(* CODESYS project Estação 5 - Sorting (2022).project

Project tree, tasks and I/O mapping:
  Device : CPX-CEC-C1-V3, Festo AG & Co. KG, order no. 3473128, version 3.5.7.37
      unmapped channels: Rotary switch
    application Application
      libraries: Standard, * (System)
      task MainTask (cyclic, interval t#20ms, priority 20) calls PLC_PRG
      program PLC_PRG [ST]
      global variables GVL
      function ATUALIZAR_VALORES [ST]
      program teste_comunicacao [ST]
      program pisca_pisca [ST]
      function SINALIZAR_QUANTIA_CORES_MODBUS [ST]
    PLC_Diagnosis : PLC-Diagnosis, Festo AG & Co. KG, version 3.5.4.1
    CPX_System : CPX_System, Festo AG & Co. KG, order no. 3473128, version 1.258
      _8DI_8DO_1 : 8DI/8DO, Festo AG & Co. KG, order no. 526257, version 1.258
          settings:  = 0;  = 1;  = 1;  = 1;  = 1;  = 0;  = 1;  = 1;  = 0;  = 0;  = 0;  = 0;  = 0;  = 0;  = 0;  = 0;  = 0;  = 0;  = 0;  = 0;  = 0;  = 0;  = 0;  = 0;  = 0;  = 0;  = 0;  = 0;  = 0;  = 0;  = 0;  = 0;  = 0;  = 0;  = 0;  = 0;  = 0;  = 0;  = 0;  = 0;
             = 0;  = 0;  = 0;  = 0;  = 0;  = 0;  = 0;  = 0;  = 0;  = 0;  = 0;  = 0;  = 0;  = 0;  = 0;  = 0;  = 0;  = 0;  = 0;  = 0;  = 0;  = 0;  = 0;  = 0;  = 0;  = 0;  = 0;  = 0;  = 0;  = 0;  = 0;  = 0;  = 0;  = 0;  = 0;  = 0;  = 0;  = 0;  = 0;  = 0;
             = 576751027668385792;  = 'PI%i.0.0.1=1';  = 'PI%i.0.1.1=1';  = 'PI%i.0.2.1=1';  = 'PI%i.1.0.1=1';  = 'PI%i.1.1.1=0';  = 'PI%i.1.4.2=1';  = 'PI%i.1.6.2=1';  = 'PI%i.6.0.1=0';  = 'PI%i.6.1.1=0';  = 'PI%i.6.2.1=0';  = 'PI%i.6.3.1=0';  = 'PI%i.6.4.1=0';  = 'PI%i.6.5.1=0';  = 'PI%i.6.6.1=0';  = 'PI%i.6.7.1=0';  = dd4a6e61;  = 6
          unmapped channels: Input 0, Output 0
      CEC_C1_V3 : CEC-C1-V3, Festo AG & Co. KG, order no. 3473128, version 1.258
          settings:  = 0;  = 150810762677760;  = 839035072;  = 65535;  = 16885952;  = 13959208;  = 1f5d2989;  = 5
      _8DI_8DO : 8DI/8DO, Festo AG & Co. KG, order no. 526257, version 1.258
          settings:  = 0;  = 1;  = 1;  = 1;  = 1;  = 0;  = 1;  = 1;  = 0;  = 0;  = 0;  = 0;  = 0;  = 0;  = 0;  = 0;  = 0;  = 0;  = 0;  = 0;  = 0;  = 0;  = 0;  = 0;  = 0;  = 0;  = 0;  = 0;  = 0;  = 0;  = 0;  = 0;  = 0;  = 0;  = 0;  = 0;  = 0;  = 0;  = 0;  = 0;
             = 0;  = 0;  = 0;  = 0;  = 0;  = 0;  = 0;  = 0;  = 0;  = 0;  = 0;  = 0;  = 0;  = 0;  = 0;  = 0;  = 0;  = 0;  = 0;  = 0;  = 0;  = 0;  = 0;  = 0;  = 0;  = 0;  = 0;  = 0;  = 0;  = 0;  = 0;  = 0;  = 0;  = 0;  = 0;  = 0;  = 0;  = 0;  = 0;  = 0;
             = 576751027668385792;  = 'PI%i.0.0.1=1';  = 'PI%i.0.1.1=1';  = 'PI%i.0.2.1=1';  = 'PI%i.1.0.1=1';  = 'PI%i.1.1.1=0';  = 'PI%i.1.4.2=1';  = 'PI%i.1.6.2=1';  = 'PI%i.6.0.1=0';  = 'PI%i.6.1.1=0';  = 'PI%i.6.2.1=0';  = 'PI%i.6.3.1=0';  = 'PI%i.6.4.1=0';  = 'PI%i.6.5.1=0';  = 'PI%i.6.6.1=0';  = 'PI%i.6.7.1=0';  = dd4a6e5f;  = 6
          unmapped channels: Input 0, Output 0
    Ethernet : Ethernet, 3S - Smart Software Solutions GmbH, version 3.5.10.0
      ModbusTCP_Slave_Device : ModbusTCP Slave Device, 3S - Smart Software Solutions GmbH, version 3.5.10.0
          unmapped channels: Inputs, Outputs
*)

// Device/Application/GVL
{attribute 'qualified_only'}
VAR_GLOBAL
	//Entradas
	//Sensores
	S_inicio 	AT %IX1.0 :BOOL; //Sensor de inicio da esteira
	S_desv_1 	AT %IX1.1 :BOOL; //Desviacdor 1 avançado
	S_rampa 	AT %IX1.2 :BOOL; //Sensor do fim da esteira
	S_desv_2	AT %IX1.3 :BOOL; //Desviacdor 2 avançado
	S_barreira 	AT %IX1.4  :BOOL; //Sensor de barreira do inicio da esteira
	S_cor 		AT %IX1.5  :BOOL; //Sesnor otico difuso para detectar peças não preta
	S_indutivo  AT %IX1.6  :BOOL; //Sensor indutivo para peças metalicas
	
	//IHM
	Start_btn 		AT	%IX2.0	:BOOL;  //Botão de start
	Stop_btn 		AT	%IX2.1	:BOOL;	//Botão de stop (NF)
	Chave 			AT	%IX2.2	:BOOL;	//Chave auto/manual
	Reset_btn 		AT	%IX2.3	:BOOL;	//Botão de reset
	I4_IHM			AT	%IX2.4	:BOOL;	//Bit de saída 4 da IHM
	I5_IHM			AT	%IX2.5	:BOOL;	//Bit de saída 5 da IHM
	I6_IHM 			AT	%IX2.6	:BOOL;	//Bit de saída 6 da IHM
	I7_IHM			AT	%IX2.7	:BOOL;	//Bit de saída 7 da IHM

//Saídas
	//Atuadorres 			
	Esteira_frente 	AT	%QX0.0	:BOOL;	//Mover a esteira para frente
	Desv_1 			AT	%QX0.1	:BOOL;	//Atua o desviador 1
	Desv_2 	 		AT	%QX0.2	:BOOL;	//Atua o desviador 2
	Stopper		 	AT	%QX0.3	:BOOL;	//Stopper recuado
	//				AT	%QX0.4	:BOOL;	
	//		 		AT	%QX0.5	:BOOL;	
	//				AT	%QX0.6	:BOOL;	
	//	     		AT	%QX0.7	:BOOL;	
	
	//IHM				
	Start_LED		AT	%QX1.0	:BOOL;	//LED do botão de start
	Reset_LED 		AT	%QX1.1	:BOOL;	//LED do botão de reset
	Q1_LED 			AT	%QX1.2	:BOOL;	//LED sinalizador Q1
	Q2_LED			AT	%QX1.3	:BOOL;	//LED sinalizador Q2
	Q4_IHM			AT	%QX1.4	:BOOL;	//Saída Q4 IHM
	Q5_IHM			AT	%QX1.5	:BOOL;	//Saída Q5 IHM
	Q6_IHM			AT	%QX1.6	:BOOL;	//Saída Q6 IHM
	Q7_IHM 			AT	%QX1.7	:BOOL;	//Saída Q7 IHM
	
//MODBUS bits
	//Entradas
	Mod_I_0_0 		AT %IX4.0 : BOOL; //Start 
	Mod_I_0_1	 	AT %IX4.1 : BOOL; //Stop
	Mod_I_0_2 		AT %IX4.2 : BOOL; //Reset
	Mod_I_0_3 		AT %IX4.3 : BOOL; //Modo entrada (DESATIVADO PARA ESSA ESTAÇÃO)
	Mod_I_0_4 		AT %IX4.4 : BOOL; //Modo saída (DESATIVADO PARA ESSA ESTAÇÃO)
	Mod_I_0_5 		AT %IX4.5 : BOOL; //Teste resposta da estação - IN 
	Mod_I_0_6 		AT %IX4.6 : BOOL; //B1 //Confirmação de leitura da informação de peça finalizada pela central
	Mod_I_0_7 		AT %IX4.7 : BOOL; //B2
	Mod_I_1_0 		AT %IX5.0 : BOOL; //B3
	Mod_I_1_1 		AT %IX5.1 : BOOL;
	Mod_I_1_2 		AT %IX5.2 : BOOL;//Confirmação de leitura da informação de peça finalizada pela central
	

	
	//Saídas
	Mod_Q_0_0 		AT %QX2.0 : BOOL; //Estação iniciada							
	Mod_Q_0_1	 	AT %QX2.1 : BOOL; // Estação parada 						
	Mod_Q_0_2 		AT %QX2.2 : BOOL; //Estação em processo										
	Mod_Q_0_3 		AT %QX2.3 : BOOL; // Modo entrada (DESATIVADO PARA ESSA ESTAÇÃO)								
	Mod_Q_0_4 		AT %QX2.4 : BOOL; // Modo saída (DESATIVADO PARA ESSA ESTAÇÃO)
	Mod_Q_0_5 		AT %QX2.5 : BOOL; // Teste resposta da estação - OUT
	
	Mod_Q_0_6 		AT %QX2.6 : BOOL; //B1 														//Sinaliza para a central que uma peça foi finalizada
	
	Mod_Q_0_7 		AT %QX2.7 : BOOL; //B2 														//BLACK B1  LSB
	Mod_Q_1_0 		AT %QX3.0 : BOOL; //B3 														//BLACK B2
	Mod_Q_1_1 		AT %QX3.1 : BOOL; 	   														//BLACK B3  MSB
	
	Mod_Q_1_2 		AT %QX3.2 : BOOL; //Sinaliza para a central que uma peça foi finalizada		//SILVER B1	LSB	
	Mod_Q_1_3 		AT %QX3.3 : BOOL;															//SILVER B2
	Mod_Q_1_4 		AT %QX3.4 : BOOL;															//SILVER B3 MSB
	
	Mod_Q_1_5 		AT %QX3.5 : BOOL;															//RED	 B1 LSB
	Mod_Q_1_6 		AT %QX3.6 : BOOL;															//RED	 B2
	Mod_Q_1_7 		AT %QX3.7 : BOOL;															//RED	 B3 MSB
	
	Mod_Q_2_0 		AT %QX4.0 : BOOL;
	Mod_Q_2_1 		AT %QX4.1 : BOOL; 
	Mod_Q_2_2 		AT %QX4.2 : BOOL;							
	Mod_Q_2_3 		AT %QX4.3 : BOOL;			
	Mod_Q_2_4 		AT %QX4.4 : BOOL;
	Mod_Q_2_5 		AT %QX4.5 : BOOL;
	Mod_Q_2_6 		AT %QX4.6 : BOOL;
	Mod_Q_2_7 		AT %QX4.7 : BOOL;
	
	

//Variáveis de lógica

	BLACK_NUM  : INT := 0;
	SILVER_NUM : INT := 0;
	RED_NUM    : INT := 0;

	B1_Modbus : BOOL;
	B2_Modbus : BOOL;
	B3_Modbus : BOOL;

	principal: BOOL;
	processo: BOOL;
	ligar_pisca :bool;
	parada: BOOL;
	passo1: BOOL;	
	passo2: BOOL;
	passo3: BOOL;
	passo4: BOOL;
	passo5: BOOL;
	passo6: BOOL;
	passo7: BOOL;
	passo8: BOOL;
	
	start: BOOL; //Start geral
	stop: BOOL;  //Stop geral
	reset: BOOL; //Reset geral
	key: BOOL; //key geral
END_VAR

// Device/Application/PLC_PRG
PROGRAM PLC_PRG
VAR
	TONInst1: Ton;
	TON_1: BOOL;
END_VAR

TONInst1(IN := TON_1, PT:= T#1S);

ATUALIZAR_VALORES();
teste_comunicacao();
pisca_pisca();

IF GVL.start  AND NOT GVL.parada AND NOT GVL.principal THEN 
	GVL.principal := TRUE;
	GVL.passo1 := TRUE;
	GVL.Q1_LED := TRUE;
	GVL.Start_LED := FALSE;
	GVL.Q7_IHM := FALSE;
	
END_IF

IF  GVL.stop THEN
	GVL.principal := FALSE;
	GVL.parada := TRUE;
	GVL.Esteira_frente :=FALSE;

	GVL.Start_LED := FALSE;
	GVL.Reset_LED := TRUE;
	GVL.Q2_LED := FALSE;
	GVL.Q1_LED := FALSE;
	gvl.ligar_pisca := FALSE;
	gvl.processo := FALSE;
	
	GVL.Q7_IHM := TRUE;
END_IF

IF GVL.reset AND NOT GVL.principal AND GVL.parada
THEN
	GVL.passo1:= FALSE;
	GVL.passo2:= FALSE;
	GVL.passo3:= FALSE;
	GVL.passo4:= FALSE;
	GVL.passo5:= FALSE;
	GVL.passo6:= FALSE;
	GVL.passo7:= FALSE;
	GVL.passo8:= FALSE;
	
	GVL.Esteira_frente :=FALSE;
	GVL.Desv_1 := FALSE;
	GVL.Desv_2 := FALSE;
	GVL.Stopper := FALSE;
	GVL.parada := FALSE;
	gvl.ligar_pisca := FALSE;
	gvl.processo := FALSE;
	GVL.Reset_LED := FALSE;
	
	GVL.B1_Modbus := FALSE;
	GVL.B2_Modbus := FALSE;
	GVL.B3_Modbus := FALSE;
	
END_IF

IF NOT GVL.principal AND NOT GVL.parada THEN 
	GVL.Start_LED := TRUE;
	GVL.Q7_IHM := TRUE;
END_IF
	

IF NOT GVL.parada THEN
		
		IF GVL.passo1 AND GVL.S_inicio THEN
			GVL.passo1 := FALSE;
			GVL.passo2 := TRUE;
			GVL.Esteira_frente := TRUE;
			gvl.ligar_pisca := TRUE;
			gvl.processo := TRUE;
			GVL.Q7_IHM := TRUE;
			GVL.B1_Modbus := FALSE;
			GVL.B2_Modbus := FALSE;
			GVL.B3_Modbus := FALSE;
		END_IF
		
		IF GVL.passo2 AND GVL.S_barreira THEN
			GVL.passo2 := FALSE;
			GVL.passo3 := TRUE;
			TON_1 := TRUE;
			
		END_IF
		
		IF GVL.passo3 AND TONInst1.Q THEN
			GVL.passo3 := FALSE;
			TON_1 := FALSE;
			GVL.Esteira_frente := FALSE;
			
			IF GVL.S_cor THEN
				IF  GVL.S_indutivo THEN
						GVL.passo7 := TRUE;	//peça prata
						GVL.B1_Modbus := FALSE;
						GVL.B2_Modbus := TRUE;
						IF NOT (gvl.SILVER_NUM = 7) THEN
							gvl.SILVER_NUM := gvl.SILVER_NUM + 1; //Soma 1 a quantidade de peças pratas processadas
						END_IF
					ELSE
						GVL.passo4 := TRUE; //Peça vermelha
						GVL.B1_Modbus := FALSE;
						GVL.B2_Modbus := FALSE;
						IF NOT (gvl.RED_NUM = 7) THEN
							gvl.RED_NUM := gvl.RED_NUM + 1; //Soma 1 a quantidade de peças vermelhas processadas 
						END_IF
				END_IF
			ELSE
				GVL.passo5 := TRUE; //peça preta
				GVL.B1_Modbus := TRUE;
				GVL.B2_Modbus := FALSE;
				IF NOT (gvl.BLACK_NUM = 7) THEN
					gvl.BLACK_NUM := gvl.BLACK_NUM + 1; //Soma 1 a quantidade de peças pretas processadas 
				END_IF
			END_IF
			GVL.Stopper := TRUE;
			GVL.Esteira_frente := TRUE;
		END_IF
		
		IF GVL.passo4 THEN
			GVL.passo4 := FALSE;
			GVL.passo7 := TRUE;
			GVL.Desv_2 := TRUE;
		END_IF
		
		IF GVL.passo5 THEN
			GVL.passo5 := FALSE;
			GVL.passo7 := TRUE;
			GVL.Desv_1 := TRUE;
		END_IF
		
		IF GVL.passo7 AND GVL.S_rampa THEN
			GVL.passo7 := FALSE;
			GVL.Esteira_frente := FALSE;
			GVL.Stopper := FALSE;
			GVL.Desv_1 := FALSE;
			GVL.Desv_2 := FALSE;
			GVL.passo1 := TRUE;
			gvl.ligar_pisca := FALSE;
			gvl.processo := FALSE;
			GVL.Q2_LED := FALSE;
			GVL.Q7_IHM := FALSE;
			GVL.Mod_Q_0_6 := TRUE; //Sianliza para a central que uma peça foi finalizada
		END_IF

END_IF

END_PROGRAM

// Device/Application/ATUALIZAR_VALORES
FUNCTION ATUALIZAR_VALORES : INT
VAR

END_VAR

GVL.Mod_Q_0_0 := GVL.principal;
GVL.Mod_Q_0_1 := GVL.parada;
GVL.Mod_Q_0_2 := gvl.processo;

//GVL.Mod_Q_0_6 := GVL.B1_Modbus;
//GVL.Mod_Q_0_7 := GVL.B2_Modbus;
//GVL.Mod_Q_1_0 := GVL.B3_Modbus;



IF GVL.Start_btn OR GVL.Mod_I_0_0 THEN  //Atualização do valor da variável de start
	GVL.start := TRUE;
	ELSE
	GVL.start := FALSE;
END_IF

IF NOT GVL.Stop_btn OR GVL.Mod_I_0_1 THEN //Atualização do valor da variável de stop
	GVL.stop := TRUE;
	ELSE
	GVL.stop := FALSE;
END_IF

IF GVL.Reset_btn OR GVL.Mod_I_0_2 THEN //Atualização do valor da variável de reset
	GVL.reset := TRUE;
	ELSE
	GVL.reset := FALSE;	
END_IF

IF GVL.Chave OR GVL.Mod_I_0_3 THEN //Atualização do valor da variável da chave
	GVL.key := TRUE;
	ELSE
	GVL.key := FALSE;
END_IF

SINALIZAR_QUANTIA_CORES_MODBUS(gvl.BLACK_NUM, "BLACK");
SINALIZAR_QUANTIA_CORES_MODBUS(gvl.SILVER_NUM, "SILVER");
SINALIZAR_QUANTIA_CORES_MODBUS(gvl.RED_NUM, "RED");

IF gvl.Mod_I_0_6 THEN //Confimação de leitura 

	gvl.Mod_Q_0_6 := FALSE;
	
	gvl.BLACK_NUM  := 0;
	gvl.RED_NUM    := 0;
	gvl.SILVER_NUM := 0;
	
END_IF

END_FUNCTION

// Device/Application/SINALIZAR_QUANTIA_CORES_MODBUS
FUNCTION SINALIZAR_QUANTIA_CORES_MODBUS : BOOL
	
VAR_INPUT
	NUM : INT;
	COLOR : WSTRING;
END_VAR
VAR
	BIT1 : BOOL;
	BIT2 : BOOL;
	BIT3 : BOOL;
END_VAR


	IF NUM = 1 OR NUM = 3 OR NUM = 5 OR NUM = 7 THEN
		BIT1 := TRUE;
	ELSE
		BIT1 := FALSE;
	END_IF



	IF NUM = 2 OR NUM = 3 OR NUM = 6 OR NUM = 7 THEN
		BIT2 := TRUE;
	ELSE
		BIT2 := FALSE;
	END_IF



	IF NUM = 4 OR NUM = 5 OR NUM = 6 OR NUM = 7 THEN
		BIT3 := TRUE;
	ELSE
		BIT3 := FALSE;
	END_IF


IF (COLOR = "BLACK") THEN
	gvl.Mod_Q_0_7 := BIT1; //LSB
	gvl.Mod_Q_1_0 := BIT2;
	gvl.Mod_Q_1_1 := BIT3; //MSB
END_IF

IF (COLOR = "SILVER") THEN
	gvl.Mod_Q_1_2 := BIT1; //LSB
	gvl.Mod_Q_1_3 := BIT2;
	gvl.Mod_Q_1_4 := BIT3; //MSB
END_IF

IF (COLOR = "RED") THEN
	gvl.Mod_Q_1_5 := BIT1; //LSB
	gvl.Mod_Q_1_6 := BIT2;
	gvl.Mod_Q_1_7 := BIT3; //MSB
END_IF

END_FUNCTION

// Device/Application/teste_comunicacao
PROGRAM teste_comunicacao
VAR
	
	TON_temp_1: TON;
	TON_1: BOOL;	

END_VAR

gvl.Mod_Q_0_5 := gvl.Mod_I_0_5;

END_PROGRAM

// Device/Application/pisca_pisca
PROGRAM pisca_pisca
VAR
	
	TON_temp_1: TON;
	TON_1: BOOL;
	TON_temp_2: TON;
	TON_2: BOOL;
	
	passo: INT;
END_VAR

TON_temp_1(IN := TON_1, PT:= T#0.2S);
TON_temp_2(IN := TON_2, PT:= T#0.2S);

IF gvl.ligar_pisca AND (passo = 0)  THEN
	TON_1 := TRUE;
	passo := 1;
END_IF

IF NOT gvl.ligar_pisca THEN
	TON_1 := FALSE;
	TON_2 := FALSE;
	GVL.Q2_LED := FALSE;
	passo := 0;
END_IF

IF TON_temp_1.Q THEN
	TON_1 := FALSE;
	TON_2 := TRUE;
	GVL.Q2_LED := TRUE;
END_IF

IF TON_temp_2.Q THEN
	TON_1 := TRUE;
	TON_2 := FALSE;
	GVL.Q2_LED := FALSE;
END_IF

END_PROGRAM
